INTERFACE I_PendingResponseMiddlewareConfig

END_INTERFACE

(* stored: Version 1.1.0.1, ProductVersion 3.1.4024.12
   Itf I_PendingResponseMiddlewareConfig: Id {84165e98-d8fc-4161-8351-d7ee8fc22df1} *)
